FUNCTION_BLOCK CmdDecode (* Basic Function Block Type *)
  (* Standard: 61499-2 *)
  (* Version 0.0, 6/4/2026, Schneider Electric, Template *)
  PACKAGE SE.Nereda;
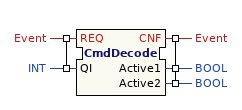
  EVENT_INPUT
    REQ WITH QI; (* Normal Execution Request *)
  END_EVENT
  EVENT_OUTPUT
    CNF WITH Active1, Active2; (* Execution Confirmation *)
  END_EVENT
  VAR_INPUT
    QI : INT; (* Input event qualifier *)
  END_VAR
  VAR_OUTPUT
    Active1 : BOOL; (* Output event qualifier *)
    Active2 : BOOL;
  END_VAR
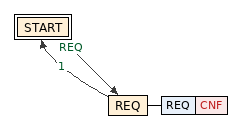
  EC_STATES
    START; (* Initial State *)
    REQ : REQ -> CNF; (* Normal execution *)
  END_STATES
  EC_TRANSITIONS
    START TO REQ := REQ;
    REQ TO START := 1;
  END_TRANSITIONS
  ALGORITHM REQ IN ST: (* Normally executed algorithm *)
;
IF QI = 1 THEN
	Active1 := TRUE;
	Active2 := FALSE;
ELSIF QI = 2 THEN
	Active1 := FALSE;
	Active2 := TRUE;
END_IF;
  END_ALGORITHM
END_FUNCTION_BLOCK
